FUNCTION_BLOCK FB_UnloadingStation IMPLEMENTS I_WorkingStation
VAR_INPUT
END_VAR
VAR_OUTPUT
END_VAR
VAR
END_VAR

PROPERTY prTableInPosition : BOOL
GET
END_GET
SET
END_SET
END_PROPERTY

{attribue 'monitoring':= call}
PROPERTY prTableRotationInterlock : BOOL
GET
END_GET
SET
END_SET
END_PROPERTY

{attribue 'monitoring':= call}
PROPERTY prTableRotationRequest : BOOL
GET
END_GET
SET
END_SET
END_PROPERTY

END_FUNCTION_BLOCK

(* stored: Version 1.1.0.1, ProductVersion 3.1.4024.15
   POU FB_UnloadingStation: Id {296f6eb6-2953-417c-abf3-86065ed0eed9}, SpecialFunc None
   Property prTableInPosition: Id {63da9327-87a5-4a03-ae22-c0f060ca43e6}
   Get Get: Id {e46b5cea-1647-4955-8397-cc47a30d7c58}
   Set Set: Id {5628a0ff-352c-4a08-8a21-2f99bb324a06}
   Property prTableRotationInterlock: Id {88e14835-694a-42c6-83c2-cd76547a82a6}
   Get Get: Id {dad85451-5c00-40c4-980f-760fb8b97cd8}
   Set Set: Id {e168513b-10c3-41ca-b98a-85bf4d086b6b}
   Property prTableRotationRequest: Id {42e13d42-38a7-4f24-9a20-9aec86822997}
   Get Get: Id {9d27c0c8-5d5b-424c-b898-aac61aa96673}
   Set Set: Id {8767d4b8-41d1-4d46-9c1a-a16455f23c2f} *)
